// TIA Portal V21 export
// export: Created 2026-05-11T00:00:00.0000000Z, ExportSetting None, DisplayName Totally Integrated Automation Portal, DisplayVersion V21, DisplayName STEP 7 Professional, DisplayVersion V21
FUNCTION "MCPVerify_FC_LAD_v3" : Void   // FC59990, LAD
TITLE = MCP LAD v3 (Lt on 安全PLC)
{ S7_Optimized_Access := 'TRUE' }
// MCP v3: Lt only — import+compile check on 安全PLC (see SKILL LAD v3)
// stored: AutoNumber false, SetENOAutomatically false
   VAR_INPUT
      CmpA : Int;
      CmpB : Int;
   END_VAR
   VAR_OUTPUT
      OutLt : Bool;
   END_VAR
BEGIN

REGION Network 1: N1-Lt
   // Lt CmpA and CmpB
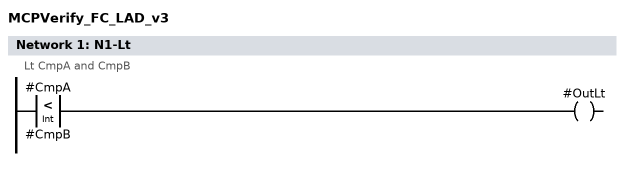
   RUNG wire#powerrail
      { S7_Templates := "SrcType := Int" } LT_Contact(in1 := #CmpA, in2 := #CmpB)
      Coil( #OutLt )
   END_RUNG
   // the same network as SCL:
   #OutLt := #CmpA < #CmpB;
END_REGION
END_FUNCTION
